RoboDK station: kr30 cnc 070419 4.rdk

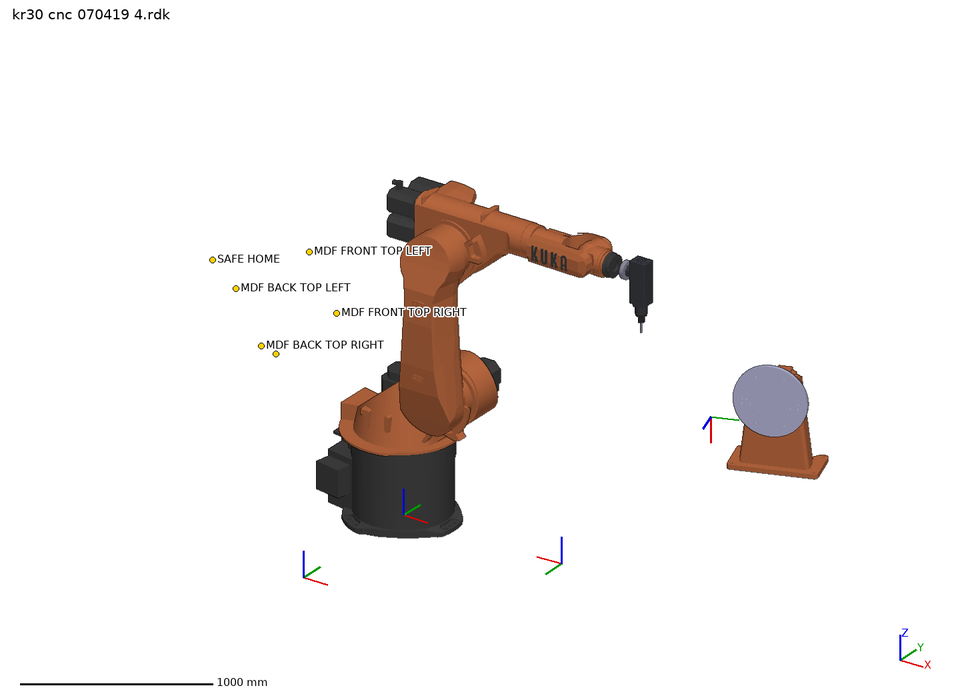
[picture v0: the station drawn from its stored meshes, robots at their saved joint values, targets as dots, program paths as lines]
Station kr30 cnc 070419 4. Poses are relative to the parent item; angles as X-Y-Z fixed-axis rotations.
  - frame GIGASHEEN 7th Axis Base at (0, 1100, 0) mm
    - robot KUKA KP1 MD250: 1 axes, payload 250 kg
        modified DH rows (alpha deg, a mm, theta deg, d mm): 0, 0, 0, 0
        base shift (1750, 1710, 820) mm, rotated rx 0 ry 90 rz -70 deg
        joint limits [-3600] to [3600]; home [0]; saved at [0]
      - frame Reference Rhino at (0, -250, 250) mm
        - object RhinoPart at (0, 0, 0) mm
  - frame GIGASHEEN Base at (0, 2000, 0) mm
    - robot GIGASHEEN (model KUKA KR 30 HA): 6 axes, payload 30 kg, reach 2033 mm, repeatability 0.05 mm, weight 665 kg
        modified DH rows (alpha deg, a mm, theta deg, d mm): 0, 0, 0, 815; -90, 350, 0, 0; 0, 850, -90, 0; -90, 145, 0, 820; 90, 0, 0, 0; -90, 0, 180, 170
        joint limits [-185, -135, -120, -350, -119, -350] to [185, 35, 158, 350, 119, 350]; home [0, -90, 90, 0, 0, 0]; saved at [0, -90, 90, 0, 0, 0]
      - tool 1/2" End Mill TCP, TCP at (337.71, -2.2, 160.57) mm, rotated rx 0 ry 90 rz 0 deg, size 415.8 x 102 x 153.6 mm
    - target MDF BACK TOP LEFT (joint target) at (-356.49, -1000.77, 1606.89) mm, rotated rx 85.17 ry 71.84 rz 47.05 deg; joints [27.716, -45.008, 102.25, 116.233, 75.695, -151.59, -681.46] of GIGASHEEN
    - target MDF FRONT TOP LEFT (joint target) at (-109.28, -692.01, 1762.49) mm, rotated rx 85.17 ry 71.84 rz 47.05 deg; joints [22.06, -21.631, 54.581, 104.768, 70.881, -126.376, -681.46] of GIGASHEEN
    - target MDF FRONT TOP RIGHT (joint target) at (-17.28, -577.35, 1389.17) mm, rotated rx 85.17 ry 71.84 rz 47.05 deg; joints [10.053, -29.315, 70.245, 98.928, 81.917, -132.341, -681.46] of GIGASHEEN
    - target MDF BACK TOP RIGHT (joint target) at (-270.04, -894.47, 1259.33) mm, rotated rx 85.17 ry 71.84 rz 47.05 deg; joints [13.787, -50.344, 113.459, 104.66, 84.215, -154.683, -681.46] of GIGASHEEN
    - target MDF STOCK DEPTH (only use z axis value) (joint target) at (-187.98, -883.66, 1230.73) mm, rotated rx 85.17 ry 71.84 rz 47.05 deg; joints [11.502, -45.737, 110.222, 102.707, 85.519, -155.78, -681.46] of GIGASHEEN
    - target SAFE HOME (joint target) at (-1094.61, -161.46, 1230.73) mm, rotated rx 85.17 ry 71.84 rz 47.05 deg; joints [11.502, -69.45, 58.776, 88.861, 76.585, -79.989, -681.46] of GIGASHEEN
  - frame Frame 4 at (1595.12, 1150.76, 505) mm, rotated rx 1.38 ry 0.62 rz -177.49 deg
  - machining project Machining Settings: C:/Users/liqui/OneDrive/Documents/GitHub/kuka-fdm/chuck.apt | rotZ(0) | rotX(0)*rotY(0) | rotz(50)
